FUNCTION_BLOCK SRFlipFlop
VAR_INPUT										//R-Dominanter RS-Baustein
	bSET: BOOL;									//Baustein-interne Set-Variable
	bRESET: BOOL;								//Baustein-interne Reset-Variable
END_VAR
VAR_OUTPUT
END_VAR
VAR
	SRFlipFlop: SR;								//Instanziierung des SR-Bausteins
END_VAR

SRFlipFlop(SET1:= bSET, RESET:= bRESET);		//Verknüpfung der Baustein-internen Variablen mit den Bausteineingängen

END_FUNCTION_BLOCK

(* stored: Version 1.1.0.1
   POU SRFlipFlop: Id {ece312e8-3366-49e8-b101-e963a64957f5}, SpecialFunc None *)
